(*********************************** G.D S.p.A. - Technical Department ***********************************
============= PROGRAM INFO ============
FOLDER:             TBD
MACHINES INVOLVED:  TBD 

============= DESCRIPTION =============
Exit unit device declaration

============= REVISIONS ===============
Date		Version	 	Author      	Description             
----------	-------		------------  	--------------------------------------------
2019/03/27 	0000.00	 	CEC 			Creation of the PRG

**********************************************************************************************************)
(*$R process_ref:= prc; $*)

PROGRAM csp_customerInterfaces

VAR
	prc:								process;
	prc_path:							STRING;
	
	Palletizer:							csp_customerInterfaces_palletizer;
	
END_VAR

VAR PERSISTENT
	CasePacker:							csp_customerInterfaces_casePacker;	
	Order:								csp_customerInterfaces_order;
	Product:							csp_customerInterfaces_product;
	Recipe:								csp_customerInterfaces_recipe;														
	Material:							ARRAY [0..14] OF csp_customerInterfaces_material;
	Mark:								csp_customerInterfaces_mark;
	NextOrder:							csp_customerInterfaces_order;	
	NextProduct:						csp_customerInterfaces_product;	
	NextRecipe:							csp_customerInterfaces_recipe;		
	NextMaterial:						ARRAY [0..14] OF csp_customerInterfaces_material;			
	MES:								csp_customerInterfaces_MES;	
		
END_VAR

_read_var_input();

_objects_manager();

IF NOT objects_running()
THEN
	RETURN;	
END_IF

_read_process_image();

_mode_manager();

CASE process_get_mode(prc) of
	MODE_ABSENT,
	MODE_INACTIVE:
		RETURN;
	MODE_TEST:
		_handle_process_test();
END_CASE

_set_runtime_properties();

(********************************* BODY *********************************)


(* CSP STATUS *)

Dock();
//CasePacker.Status.Online := machine_is_operational(csp.mch); 
//CasePacker.Status.Job := csp_main_brand.p_carton_format;
//CasePacker.Status.NextJob := // need to figure out next job
//CasePacker.Status.Running := machine_is_running(csp.mch);

//**************Variables controlled in csp_main_phaseManager.variables_update******************************

(*CasePacker.Status.Faulted.Main := machine_is_stopped(csp.mch)
									AND csp_main_interface.alarm_id_from_python <> 431 // CYCLE STOP FOR CASE SIDE
									AND csp_main_interface.alarm_id_from_python <> 769; // CYCLE STOP FOR TRANSFER SIDE*)
//CasePacker.Status.Faulted.CaseBlanks := csp_case_feed_magazine.AML_Faulted;

//CasePacker.Status.RunOut := csp_main_motorization.empty_command;
//CasePacker.Status.RunOutComplete := message_is_on(csp_case_virtualMaster.runout_complete);

//CasePacker.Status.Rate.Target := LREAL_TO_INT(csp_main_motorization_manager.motm.actual_velocity_setpoint);
//CasePacker.Status.Rate.Actual := LREAL_TO_INT(csp_main_motorization_manager.motm.actual_velocity);

//CasePacker.Status.Stop.AutoReason := csp_main_interface.alarm_id; 
//CasePacker.Status.Stop.Estop := machine_is_stop_emergency_active(csp.mch);
//CasePacker.Status.Stop.Guard := NOT safety_integrated_series_is_safely_closed(csp_case_main_safety_guards.sis) OR NOT safety_integrated_series_is_safely_closed(csp_transfer_main_safety_guards.sis);
//CasePacker.Status.Stop.Operator := message_is_on(csp_case_main_services_pushbuttons.stop_dchk.alarm_asm.message);

//CasePacker.Status.Starved.CaseBlanks := message_is_on(csp_case_feed_magazine_level_zonemin.magazine_level_zone_min_wem);
//CasePacker.Status.Starved.Glue := NOT digital_input_is_active(csp_case_glue_hotmelt.level_ok_di);
//CasePacker.Status.Starved.Labels :=
//CasePacker.Status.Starved.Units := csp_transfer_infeed_clamp.min_prime;

//CasePacker.Status.Blocked.Downstream := message_is_on(csp_case_discharge_reject_sensors.downstream_backup_hold_aem);
//CasePacker.Status.Blocked.Reject := message_is_on(csp_case_discharge_reject_sensors.consecutive_blocked_reject_aem);
//CasePacker.Status.Blocked.Waste := message_is_on(csp_transfer_crosspusher_reject.backup_di_dchk.alarm_asm.message);

//CasePacker.Labels.Consumed:=


(************************************************************************)

_handle_messages();

_write_output();

ACTION _handle_messages:
;
END_ACTION

ACTION _handle_process_test:
;
END_ACTION

ACTION _mode_manager:
IF process_mode_req_is_pending(prc)
THEN
    process_apply_mode_req_first_step(prc);
    CASE process_get_mode(prc) OF
        MODE_TO_ABSENT:
			;
        MODE_TO_INACTIVE:
			;
        MODE_TO_TEST:
			;
        MODE_TO_OPERATIONAL:
			;
    END_CASE
    process_apply_mode_req_second_step(prc);
END_IF
END_ACTION

ACTION _objects_manager:
IF objects_initialization()
THEN
	process_init(
		object_name					:= 'csp_customerInterfaces.prc', 
		machine						:= csp.mch, 
		CONVERSION_this				:= prc);
		
	prc_path 						:= process_get_path(prc);
END_IF

IF objects_running()
THEN
	process_cycle(prc);
END_IF
END_ACTION

ACTION _read_process_image:
;
END_ACTION

ACTION _read_var_input:
;
END_ACTION

ACTION _set_runtime_properties:
;
END_ACTION

ACTION _write_output:
;
END_ACTION

ACTION Dock:
//Flexlink to AMR Dock 1
CasePacker.Dock[1].DropAvailable:= csp_case_feed_magazine.Flexlink_to_AMR_DropAvailable_1;
CasePacker.Dock[1].PickAvailable:= csp_case_feed_magazine.Flexlink_to_AMR_PickAvailable_1; 
CasePacker.Dock[1].Active:= csp_case_feed_magazine.Flexlink_to_AMR_Active_1;
CasePacker.Dock[1].EntryAck:= csp_case_feed_magazine.Flexlink_to_AMR_EntryAck_1;
CasePacker.Dock[1].EntryOK:= csp_case_feed_magazine.Flexlink_to_AMR_EntryOK_1;

RAJ_to_Flexlink[3].0:= CasePacker.Dock[1].EntryReq;
RAJ_to_Flexlink[3].1:= CasePacker.Dock[1].AmrExited;

//Flexlink to AMR Dock 2
CasePacker.Dock[2].DropAvailable:= csp_case_feed_magazine.Flexlink_to_AMR_DropAvailable_2;
CasePacker.Dock[2].PickAvailable:= csp_case_feed_magazine.Flexlink_to_AMR_PickAvailable_2; 
CasePacker.Dock[2].Active:= csp_case_feed_magazine.Flexlink_to_AMR_Active_2;
CasePacker.Dock[2].EntryAck:= csp_case_feed_magazine.Flexlink_to_AMR_EntryAck_2;
CasePacker.Dock[2].EntryOK:= csp_case_feed_magazine.Flexlink_to_AMR_EntryOK_2;

RAJ_to_Flexlink[3].2:= CasePacker.Dock[2].EntryReq;
RAJ_to_Flexlink[3].3:= CasePacker.Dock[2].AmrExited;

//Flexlink to AMR Dock 3
CasePacker.Dock[3].DropAvailable:= csp_case_feed_magazine.Flexlink_to_AMR_DropAvailable_3;
CasePacker.Dock[3].PickAvailable:= csp_case_feed_magazine.Flexlink_to_AMR_PickAvailable_3; 
CasePacker.Dock[3].Active:= csp_case_feed_magazine.Flexlink_to_AMR_Active_3;
CasePacker.Dock[3].EntryAck:= csp_case_feed_magazine.Flexlink_to_AMR_EntryAck_3;
CasePacker.Dock[3].EntryOK:= csp_case_feed_magazine.Flexlink_to_AMR_EntryOK_3;

RAJ_to_Flexlink[3].4:= CasePacker.Dock[3].EntryReq;
RAJ_to_Flexlink[3].5:= CasePacker.Dock[3].AmrExited;
END_ACTION

END_PROGRAM

(* stored: Version 1.1.0.1, ProductVersion 3.1.4024.3
   POU csp_customerInterfaces: Id {69c39abf-9e2c-0e5e-3b1a-84f4916da600}, SpecialFunc None
   Action _handle_messages: Id {56a52f55-57ee-0a7e-1770-561bd0f306e3}
   Action _handle_process_test: Id {a9ac4e0f-a9e6-0ec8-34f4-11eccba2a5c1}
   Action _mode_manager: Id {d36ca099-46c3-0a12-2c5c-07bd01e102bb}
   Action _objects_manager: Id {f3afc0e1-13e5-0c9b-3636-2ced0573a774}
   Action _read_process_image: Id {422738ef-5109-023a-095f-31a07bcadb8e}
   Action _read_var_input: Id {cf9735d3-d2cc-0213-1c0b-5fc65620c6f5}
   Action _set_runtime_properties: Id {5266b757-0fa1-0a46-24eb-cbb35a1aa227}
   Action _write_output: Id {0fc51ccb-b939-017c-09d4-1737f7418ba7}
   Action Dock: Id {f0be1169-aa58-0903-34df-38822ff4cf83} *)
